FUNCTION_BLOCK FB_Integrate
VAR_INPUT
	run : BOOL 	:= TRUE;	// Set true for running integration
	in 	: REAL;				// integrated value
	K 	: REAL 	:= 1.0;		// factor
	RST	: BOOL  :=FALSE;	// set true for reinitialization
	inStart : REAL :=0; 		// start value
END_VAR

VAR_OUTPUT
	out 	: REAL;
END_VAR

VAR
	in_last : REAL;
	init: BOOL;
	last: TIME;
	tx: TIME;
END_VAR

(*read system time *)
tx := TIME();

//reset integration
IF RST = TRUE THEN
	init := FALSE;	
	out := inStart;
END_IF

IF NOT init THEN	//init last_in and skip integration for the first run
	init := TRUE;
	in_last := in;
	out := inStart;
ELSIF run THEN
	out := (in + in_last) * 0.5E-3 * TIME_TO_REAL(tx-last) * K + out;	//integration with trapezoidal rule
	in_last := in;
END_IF;
last := tx;	//save last time

END_FUNCTION_BLOCK

(* stored: Version 1.1.0.1, ProductVersion 3.1.4022.7
   POU FB_Integrate: Id {6780b537-a2b0-444b-acad-09d50de8242d}, SpecialFunc None *)
